PROGRAM fbGetCurrentScheduleLine

VAR_OUTPUT
	arrRecords: ST_ScheduleStruct;
	sSeverity: WSTRING(255);
	bError :BOOL;

	iLines: UDINT;
END_VAR
VAR
	STProgram: ST_ProgramStruct;
	now : TIMESTRUCT;
	nowMinutes : LINT;
	
	previousMinute: LINT;
	
	fbTON: TON := (PT := TIME#10S0MS);

	

	
	fbPLCDBRead : FB_PLCDBRead(sNetID:='',tTimeout:=T#5S);
	fbSqlCommand : FB_SQLCommand(sNetID := '', tTimeout := T#5S);
	
	
	intTime: DINT;
	todTime: TOD;

	sCmd: STRING(255):='SELECT * FROM [Schedule] ORDER BY [Sequence] ASC';

	dIntSqlResult: DINT;
	fbSQLDatabase: FB_SQLDatabase(sNetID:='', tTimeout:=T#10S);
	fbSQLResult: FB_SQLResult(sNetID:='', tTimeout:=T#10S);
	result: I_TcResultEvent;


	iState: INT;
END_VAR

//Build command



sCmd :=CONCAT('SELECT * FROM [Schedule] WHERE [Sequence]=',LINT_TO_STRING(GVL.ScheduleSequence));

//State machine
CASE iState OF
0:
//IDLE
fbTON(PT := TIME#3S0MS);
IF fbTON.Q=TRUE THEN
	iState:=1;
	fbTON.IN:=FALSE;
	bError := FALSE; 
ELSE
	fbTON.IN:=TRUE;
END_IF
//Connect
1:
	IF fbSqlDatabase.Connect(1) THEN
		IF fbSqlDatabase.bError THEN
			iState := 255;
			result := fbSqlDatabase.ipTcResultEvent;
			sSeverity := result.Text;
			bError := TRUE; 		
		ELSE
			//If sucessful, point the connection to the sql command function
			fbSqlDatabase.CreateCmd(ADR(fbSqlCommand));
			iState := 2;
		END_IF
	END_IF
2:
//Send the sql command
	IF fbSQLCommand.ExecuteDataReturn(ADR(sCmd), SIZEOF(sCmd), ADR(fbSqlResult)) THEN
		IF fbSQLCommand.bError THEN
			iState := 255;
			result := fbSQLCommand.ipTcResultEvent;
			sSeverity := result.Text;
			bError := TRUE;
		ELSE
			iState := 3; 
			iLines:=fbSqlResult.nDataCount;
		END_IF
	END_IF
		
3:
//Read the sql result
	IF fbSqlResult.Read(0, 1, ADR(arrRecords), SIZEOF(arrRecords), TRUE, TRUE) THEN
		IF fbSqlResult.bError THEN
			result := fbSqlResult.ipTcResultEvent;
			sSeverity := result.Text;
			iState:=255;
			bError := TRUE;
		ELSE 
			iState:=4;
			
			result := fbSqlResult.ipTcResultEvent;
			sSeverity := result.Text;
		END_IF
	

	END_IF
4:
	IF 	fbSqlDatabase.Disconnect() THEN
		bError := FALSE;
		iState:=0;
	END_IF
255:
	IF 	fbSqlDatabase.Disconnect() THEN
		iState:=0;	
		bError := TRUE;
		result := fbSqlResult.ipTcResultEvent;
		sSeverity := result.Text;

	END_IF
	
END_CASE

END_PROGRAM

(* stored: Version 1.1.0.1, ProductVersion 3.1.4022.16
   POU fbGetCurrentScheduleLine: Id {1e1b130a-77dd-4540-8514-31c58d8f8e6a}, SpecialFunc None *)
